// TIA Portal V18 export
TYPE "SubProcessParameterP050_ShW"
// stored: IsFailsafeCompliant false
   STRUCT
      SubProcessParameter : Struct
         press_force_max_value : Struct
            press_force_max_value : Real;
            press_force_max_result : Int;
            press_force_max_NG_code : String[9];
         END_STRUCT;
         displacement_max_value : Struct
            displacement_max_value : Real;
            displacement_max_result : Int;
            displacement_max_NG_code : String[9];
         END_STRUCT;
      END_STRUCT;
   END_STRUCT;
END_TYPE
